(* CoDeSys 2.3 export: ST_LOAD_CAL.EXP *)

(* Data type *)
TYPE ST_LOAD_CAL :
STRUCT
	K : REAL;
	C : REAL;
END_STRUCT
END_TYPE
